PROGRAM MAIN
VAR
	fbStateExample: StateExample;
END_VAR

fbStateExample();

END_PROGRAM

(* stored: Version 1.1.0.1, ProductVersion 3.1.4024.3
   POU MAIN: Id {0de54b69-b289-400f-9b97-65c47cc250c0}, SpecialFunc None *)
